// TwinCAT 3 PLC project Programma
// ProgramVersion: 3.1.4024.0
// libraries:
//   Tc2_Standard, * (Beckhoff Automation GmbH)
//   Tc2_System, * (Beckhoff Automation GmbH)
//   Tc3_Module, * (Beckhoff Automation GmbH)
// project tree:
//   GVLs/ GVL.TcGVL
//   / PlcTask.TcTTO
//   POUs/ MAIN.TcPOU
// real-time tasks:
//   TASK PlcTask: cycle T#10ms, priority 20, ADS port 350
// I/O:
//   DEVICE Device 2 (EtherCAT), AmsNetId 192.168.178.141.3.1
//     Term 1 (EK1100) [EK1100 EtherCAT Coupler (2A E-Bus)]
//       Term 2 (EL1008) [EL1008 8Ch. Dig. Input 24V, 3ms]
//       Term 3 (EL1008) [EL1008 8Ch. Dig. Input 24V, 3ms]
//       Term 4 (EL2004) [EL2004 4Ch. Dig. Output 24V, 0.5A]
//       Term 5 (EL9011) [EL9011 End Terminal]
// variable links:
//   Programma/Programma Instance <-> Device 2 (EtherCAT)/Term 1 (EK1100)/Term 2 (EL1008)
//     PlcTask Inputs/GVL.sensor{1..4} <-> Channel {1..4}/Input  (4 links)
//   Programma/Programma Instance <-> Device 2 (EtherCAT)/Term 1 (EK1100)/Term 4 (EL2004)
//     PlcTask Outputs/GVL.Motor1 <-> Channel 1/Output
//     PlcTask Outputs/GVL.Motor2 <-> Channel 2/Output
//     PlcTask Outputs/GVL.Motor3 <-> Channel 3/Output

CONFIGURATION Programma
    RESOURCE PLC ON TwinCAT3
        TASK PlcTask(INTERVAL := T#10ms, PRIORITY := 20);
        PROGRAM MAIN WITH PlcTask : MAIN;
    END_RESOURCE
END_CONFIGURATION

// ---- GVLs/GVL.TcGVL
{attribute 'qualified_only'}
VAR_GLOBAL
	IN_motor1 AT %I* :BOOL;
	IN_motor2 AT %I* :BOOL;
	IN_motor3 AT %I* :BOOL;
	Sensor4 AT %I* :BOOL; // wordt niet gebruikt
	RobotIn AT %I* :BOOL;
	Startknop AT %I* :BOOL;
		
	Motor1 AT %Q* :BOOL;
	Motor2 AT %Q* :BOOL;
	Motor3 AT %Q* :BOOL;
	RobotUit AT %Q* :BOOL;
	
END_VAR

// ---- POUs/MAIN.TcPOU
PROGRAM MAIN
VAR
	Step				: UINT := 0;
	Timer_output				: TON;
	Timer_motor					: TON;
END_VAR

Timer_output ();
Timer_motor ();

CASE Step OF
	0: // Startknop indrukken voor het beginnen van het systeem
 		IF gvl.Startknop = TRUE THEN 
			Step 					  	:= 10;
 		END_IF;
		 
	10: // Signaal naar robot, controleren componenten en componenten in houders plaatsten.
		gvl.RobotUit := TRUE;
		Timer_output(IN:=TRUE, PT:=T#2S); // reset output.
			
		IF Timer_output.Q = TRUE THEN
			Timer_output(IN:=FALSE);
			gvl.RobotUit := FALSE;
			Step 						:= 20;
		END_IF
	
	20: // Robot heeft componenten gecontroleerd en alles is aanwezig. Motor 1 aanzetten.
		IF gvl.IN_motor1 = TRUE THEN
			gvl.Motor1 := TRUE;
			Timer_motor (IN:=TRUE, PT:=T#10S); // tijd voor aandraaien onderdeel.
			step 						:= 30;
		END_IF
		
	30: // Wachten op montage		
		IF Timer_motor.Q = TRUE THEN
			Timer_motor (IN:=FALSE);
			gvl.Motor1 := FALSE;
			gvl.RobotUit := TRUE;
			Timer_output(IN:=TRUE, PT:=T#2S); // reset output.
			step						:= 40;
		END_IF
		
			
	40: // reseten output
		IF Timer_output.Q = TRUE THEN
			Timer_output(IN:=FALSE);
			gvl.RobotUit := FALSE;
			step 						:= 50;
		END_IF
			 

	50: // Motor 2 aanzetten.
		IF gvl.IN_motor1 = TRUE THEN
			gvl.Motor1 := TRUE;
			Timer_motor (IN:=TRUE, PT:=T#10S); // tijd voor aandraaien onderdeel.
			step						:= 60;
		END_IF;
	
	60: // Wachten op 2de monatge
		IF Timer_motor.Q = TRUE THEN
			Timer_motor (IN:=FALSE);
			gvl.Motor1 := FALSE;
			gvl.RobotUit := TRUE;
			Timer_output(IN:=TRUE, PT:=T#2S); // reset output.
			step						:=70;
		END_IF
		
			
	70: // resetten output
			IF Timer_output.Q = TRUE THEN
				Timer_output(IN:=FALSE);
				gvl.RobotUit := FALSE;
				step 					:= 80;
			END_IF
	
	80: // Motor 3 aanzetten.
		IF gvl.IN_motor1 = TRUE THEN
			gvl.Motor1 := TRUE;
			Timer_motor (IN:=TRUE, PT:=T#10S); // tijd voor aandraaien onderdeel.
			step 						:= 90;
		END_IF;
	
	90: // Wachten op 3de monatge		
		IF Timer_motor.Q = TRUE THEN
			Timer_motor (IN:=FALSE);
			gvl.Motor1 := FALSE;
			gvl.RobotUit := TRUE;
			Timer_output(IN:=TRUE, PT:=T#2S); // reset output.
			step						:=100;
		END_IF
		
			
	100: // reseten output
		IF Timer_output.Q = TRUE THEN
			Timer_output(IN:=FALSE);
			gvl.RobotUit := FALSE;
			step 						:= 110;
		END_IF
		
	110: // Alles geassembleerd.
		step 							:= 0;
		
			
END_CASE

END_PROGRAM
